// TwinCAT 3 PLC project ProyMain
// ProgramVersion: 3.1.4024.0
// libraries:
//   Tc2_Standard, * (Beckhoff Automation GmbH)
//   Tc2_System, * (Beckhoff Automation GmbH)
//   Tc3_Module, * (Beckhoff Automation GmbH)
// project tree:
//   / PlcTask.TcTTO (not stored)
//   POUs/ MAIN.TcPOU

// ---- POUs/MAIN.TcPOU
PROGRAM MAIN
VAR
	
	Pulsador AT %I*: BOOL;
	Lampara AT %Q*: BOOL;

END_VAR

Pulsador := Lampara;

END_PROGRAM
